// TwinCAT 3 PLC project KbRail
// ProgramVersion: 3.1.4022.7
// libraries:
//   Tc2_MC2, * (Beckhoff Automation GmbH)
//   Tc2_Standard, * (Beckhoff Automation GmbH)
//   Tc2_System, * (Beckhoff Automation GmbH)
//   Tc3_Module, * (Beckhoff Automation GmbH)
// project tree:
//   DUTs/ ST_AxisGroup.TcDUT
//   / PlcTask.TcTTO
//   POUs/ MAIN.TcPOU
// real-time tasks:
//   TASK PlcTask: cycle T#10ms, priority 20, ADS port 350
// motion (NC):
//   TASK NC-Task 1 SAF: cycle T#2ms, priority 4, ADS port 501
//   TASK NC-Task 1 SVB: cycle T#10ms, priority 8, ADS port 511
//   AXIS Axis 1 (id 1)
//     Dynamic: AccelerationMaximum=0.6, DecelerationMaximum=0.6, Acceleration=0.59988, Deceleration=0.59988, Jerk=1.19952, DelayTime=0.008
//     Velo: Maximum=0.1
//     OtherSettings: AllowMotionCmdToSlave=true
//     encoder EncType=29
//       EncPara: ScaleFactorNumerator=1e-06, MaxCount=#xffffffff, EvaluationDirection=2
//         SoftEndMinControl: Enable=true, Range=5
//         Inc: RefSoftSyncMask=#x0000ffff
//     drive DrvType=24
//       DrvPara: Inverse=true
//         Analog: VeloReferenz=0.4, ScaleFactorActTorque=0.1
//         TimeComp: TaskDelayCycles=1
//     controller CtrType=1
//       CtrPara: PriorControlFactor=1
//         PosDiffControl: Range=0.2
//         Observer: BandWidth=20
//   AXIS Axis 2 (id 2)
//     Dynamic: AccelerationMaximum=0.6, DecelerationMaximum=0.6, Acceleration=0.59988, Deceleration=0.59988, Jerk=1.19952, DelayTime=0.008
//     Velo: Maximum=0.1
//     OtherSettings: AllowMotionCmdToSlave=true
//     encoder EncType=29
//       EncPara: ScaleFactorNumerator=1e-06, MaxCount=#xffffffff
//         SoftEndMinControl: Enable=true, Range=5
//         Inc: RefSoftSyncMask=#x0000ffff
//     drive DrvType=24
//       DrvPara: Inverse=true
//         Analog: VeloReferenz=0.4, ScaleFactorActTorque=0.1
//         TimeComp: TaskDelayCycles=1
//     controller CtrType=1
//       CtrPara: PriorControlFactor=1
//         PosDiffControl: Range=0.2
//         Observer: BandWidth=20
//   AXIS Axis 3 (id 3)
//     General: UnitName=nm
//     Dynamic: AccelerationMaximum=0.6, DecelerationMaximum=0.6, Acceleration=0.59988, Deceleration=0.59988, Jerk=1.19952, DelayTime=0.008
//     Velo: Maximum=0.1
//     OtherSettings: AllowMotionCmdToSlave=true
//     encoder EncType=29
//       EncPara: ScaleFactorNumerator=1e-06, MaxCount=#xffffffff
//         SoftEndMinControl: Enable=true, Range=6.25
//         Inc: RefSoftSyncMask=#x0000ffff
//     drive DrvType=24
//       DrvPara: Inverse=true
//         Analog: VeloReferenz=0.4, ScaleFactorActTorque=0.1
//         TimeComp: TaskDelayCycles=1
//     controller CtrType=1
//       CtrPara: PriorControlFactor=1
//         PosDiffControl: Range=0.2
//         Observer: BandWidth=20
//   AXIS Axis 4 (id 4)
//     General: UnitName=nm
//     Dynamic: AccelerationMaximum=0.6, DecelerationMaximum=0.6, Acceleration=0.59988, Deceleration=0.59988, Jerk=1.19952, DelayTime=0.008
//     Velo: Maximum=1
//     OtherSettings: AllowMotionCmdToSlave=true
//     encoder EncType=29
//       EncPara: ScaleFactorNumerator=1e-06, MaxCount=#xffffffff
//         SoftEndMinControl: Enable=true, Range=5.5
//         Inc: RefSoftSyncMask=#x0000ffff
//     drive DrvType=24
//       DrvPara: Inverse=true
//         Analog: VeloReferenz=0.4, ScaleFactorActTorque=0.1
//         TimeComp: TaskDelayCycles=1
//     controller CtrType=1
//       CtrPara: PriorControlFactor=1
//         PosDiffControl: Range=0.2
//         Observer: BandWidth=20
// I/O:
//   DEVICE Device 1 (EtherCAT), AmsNetId 192.168.1.82.3.1
//     Term 12 (EK1100) [EK1100 EtherCAT Coupler (2A E-Bus)]
//       E1(EL7041) [EL7041 1Ch. Stepper motor output stage (50V, 5A)]
//       E2(EL5042) [EL5042 2Ch. BiSS-C Encoder]
//       E3(EL7041) [EL7041 1Ch. Stepper motor output stage (50V, 5A)]
//       E4(EL3202-0010)
//       E5(EL7041) [EL7041 1Ch. Stepper motor output stage (50V, 5A)]
//       E6(EL5042) [EL5042 2Ch. BiSS-C Encoder]
//       E7(EL7041) [EL7041 1Ch. Stepper motor output stage (50V, 5A)]
//       E8(EL3202-0010)
//       Term 23 (EL9011) [EL9011 End Terminal]
// variable links:
//   NC-Task 1 SAF/Axes/Axis 1 <-> Device 1 (EtherCAT)/Term 12 (EK1100)/E1(EL7041)
//     Drive/Inputs/In/nState1 @bit 3 <-> STM Status/Status/Error
//     Drive/Inputs/In/nState1 @bit 5 <-> STM Status/Status/Moving negative
//     Drive/Inputs/In/nState1 @bit 4 <-> STM Status/Status/Moving positive
//     Drive/Inputs/In/nState1 @bit 1 <-> STM Status/Status/Ready
//     Drive/Inputs/In/nState1 <-> STM Status/Status/Ready to enable
//     Drive/Inputs/In/nState1 @bit 6 <-> STM Status/Status/Torque reduced
//     Drive/Inputs/In/nState1 @bit 2 <-> STM Status/Status/Warning
//     Drive/Inputs/In/nState2 @bit 5 <-> STM Status/Status/Sync error
//     Drive/Inputs/In/nState2 @bit 7 <-> STM Status/Status/TxPDO Toggle
//     Drive/Inputs/In/nState4 @bit 1 <-> WcState/InputToggle
//     Drive/Inputs/In/nState4 <-> WcState/WcState
//     Drive/Outputs/Out/nCtrl1 <-> STM Control/Control/Enable
//     Drive/Outputs/Out/nCtrl1 @bit 2 <-> STM Control/Control/Reduce torque
//     Drive/Outputs/Out/nCtrl1 @bit 1 <-> STM Control/Control/Reset
//     Drive/Outputs/Out/nDataOut2[0] <-> STM Velocity/Velocity
//   NC-Task 1 SAF/Axes/Axis 1 <-> Device 1 (EtherCAT)/Term 12 (EK1100)/E2(EL5042)
//     Enc/Inputs/In/nComState @bit 1 <-> WcState/InputToggle
//     Enc/Inputs/In/nComState <-> WcState/WcState
//     Enc/Inputs/In/nDataIn1 <-> FB Inputs Channel 1/Position
//     Enc/Inputs/In/nState1 @bit 12 <-> FB Inputs Channel 1/Status/Diag
//     Enc/Inputs/In/nState1 @bit 1 <-> FB Inputs Channel 1/Status/Error
//     Enc/Inputs/In/nState1 @bit 14 <-> FB Inputs Channel 1/Status/Input cycle counter
//     Enc/Inputs/In/nState1 @bit 2 <-> FB Inputs Channel 1/Status/Ready
//     Enc/Inputs/In/nState1 @bit 13 <-> FB Inputs Channel 1/Status/TxPDO State
//     Enc/Inputs/In/nState1 <-> FB Inputs Channel 1/Status/Warning
//   NC-Task 1 SAF/Axes/Axis 2 <-> Device 1 (EtherCAT)/Term 12 (EK1100)/E2(EL5042)
//     Enc/Inputs/In/nComState @bit 1 <-> WcState/InputToggle
//     Enc/Inputs/In/nComState <-> WcState/WcState
//     Enc/Inputs/In/nDataIn1 <-> FB Inputs Channel 2/Position
//     Enc/Inputs/In/nState1 @bit 12 <-> FB Inputs Channel 2/Status/Diag
//     Enc/Inputs/In/nState1 @bit 1 <-> FB Inputs Channel 2/Status/Error
//     Enc/Inputs/In/nState1 @bit 14 <-> FB Inputs Channel 2/Status/Input cycle counter
//     Enc/Inputs/In/nState1 @bit 2 <-> FB Inputs Channel 2/Status/Ready
//     Enc/Inputs/In/nState1 @bit 13 <-> FB Inputs Channel 2/Status/TxPDO State
//     Enc/Inputs/In/nState1 <-> FB Inputs Channel 2/Status/Warning
//   NC-Task 1 SAF/Axes/Axis 2 <-> Device 1 (EtherCAT)/Term 12 (EK1100)/E3(EL7041)
//     Drive/Inputs/In/nState1 @bit 3 <-> STM Status/Status/Error
//     Drive/Inputs/In/nState1 @bit 5 <-> STM Status/Status/Moving negative
//     Drive/Inputs/In/nState1 @bit 4 <-> STM Status/Status/Moving positive
//     Drive/Inputs/In/nState1 @bit 1 <-> STM Status/Status/Ready
//     Drive/Inputs/In/nState1 <-> STM Status/Status/Ready to enable
//     Drive/Inputs/In/nState1 @bit 6 <-> STM Status/Status/Torque reduced
//     Drive/Inputs/In/nState1 @bit 2 <-> STM Status/Status/Warning
//     Drive/Inputs/In/nState2 @bit 5 <-> STM Status/Status/Sync error
//     Drive/Inputs/In/nState2 @bit 7 <-> STM Status/Status/TxPDO Toggle
//     Drive/Inputs/In/nState4 @bit 1 <-> WcState/InputToggle
//     Drive/Inputs/In/nState4 <-> WcState/WcState
//     Drive/Outputs/Out/nCtrl1 <-> STM Control/Control/Enable
//     Drive/Outputs/Out/nCtrl1 @bit 2 <-> STM Control/Control/Reduce torque
//     Drive/Outputs/Out/nCtrl1 @bit 1 <-> STM Control/Control/Reset
//     Drive/Outputs/Out/nDataOut2[0] <-> STM Velocity/Velocity
//   NC-Task 1 SAF/Axes/Axis 3 <-> Device 1 (EtherCAT)/Term 12 (EK1100)/E5(EL7041)
//     Drive/Inputs/In/nState1 @bit 3 <-> STM Status/Status/Error
//     Drive/Inputs/In/nState1 @bit 5 <-> STM Status/Status/Moving negative
//     Drive/Inputs/In/nState1 @bit 4 <-> STM Status/Status/Moving positive
//     Drive/Inputs/In/nState1 @bit 1 <-> STM Status/Status/Ready
//     Drive/Inputs/In/nState1 <-> STM Status/Status/Ready to enable
//     Drive/Inputs/In/nState1 @bit 6 <-> STM Status/Status/Torque reduced
//     Drive/Inputs/In/nState1 @bit 2 <-> STM Status/Status/Warning
//     Drive/Inputs/In/nState2 @bit 5 <-> STM Status/Status/Sync error
//     Drive/Inputs/In/nState2 @bit 7 <-> STM Status/Status/TxPDO Toggle
//     Drive/Inputs/In/nState4 @bit 1 <-> WcState/InputToggle
//     Drive/Inputs/In/nState4 <-> WcState/WcState
//     Drive/Outputs/Out/nCtrl1 <-> STM Control/Control/Enable
//     Drive/Outputs/Out/nCtrl1 @bit 2 <-> STM Control/Control/Reduce torque
//     Drive/Outputs/Out/nCtrl1 @bit 1 <-> STM Control/Control/Reset
//     Drive/Outputs/Out/nDataOut2[0] <-> STM Velocity/Velocity
//   NC-Task 1 SAF/Axes/Axis 3 <-> Device 1 (EtherCAT)/Term 12 (EK1100)/E6(EL5042)
//     Enc/Inputs/In/nComState @bit 1 <-> WcState/InputToggle
//     Enc/Inputs/In/nComState <-> WcState/WcState
//     Enc/Inputs/In/nDataIn1 <-> FB Inputs Channel 1/Position
//     Enc/Inputs/In/nState1 @bit 12 <-> FB Inputs Channel 1/Status/Diag
//     Enc/Inputs/In/nState1 @bit 1 <-> FB Inputs Channel 1/Status/Error
//     Enc/Inputs/In/nState1 @bit 14 <-> FB Inputs Channel 1/Status/Input cycle counter
//     Enc/Inputs/In/nState1 @bit 2 <-> FB Inputs Channel 1/Status/Ready
//     Enc/Inputs/In/nState1 @bit 13 <-> FB Inputs Channel 1/Status/TxPDO State
//     Enc/Inputs/In/nState1 <-> FB Inputs Channel 1/Status/Warning
//   NC-Task 1 SAF/Axes/Axis 4 <-> Device 1 (EtherCAT)/Term 12 (EK1100)/E6(EL5042)
//     Enc/Inputs/In/nComState @bit 1 <-> WcState/InputToggle
//     Enc/Inputs/In/nComState <-> WcState/WcState
//     Enc/Inputs/In/nDataIn1 <-> FB Inputs Channel 2/Position
//     Enc/Inputs/In/nState1 @bit 12 <-> FB Inputs Channel 2/Status/Diag
//     Enc/Inputs/In/nState1 @bit 1 <-> FB Inputs Channel 2/Status/Error
//     Enc/Inputs/In/nState1 @bit 14 <-> FB Inputs Channel 2/Status/Input cycle counter
//     Enc/Inputs/In/nState1 @bit 2 <-> FB Inputs Channel 2/Status/Ready
//     Enc/Inputs/In/nState1 @bit 13 <-> FB Inputs Channel 2/Status/TxPDO State
//     Enc/Inputs/In/nState1 <-> FB Inputs Channel 2/Status/Warning
//   NC-Task 1 SAF/Axes/Axis 4 <-> Device 1 (EtherCAT)/Term 12 (EK1100)/E7(EL7041)
//     Drive/Inputs/In/nState1 @bit 3 <-> STM Status/Status/Error
//     Drive/Inputs/In/nState1 @bit 5 <-> STM Status/Status/Moving negative
//     Drive/Inputs/In/nState1 @bit 4 <-> STM Status/Status/Moving positive
//     Drive/Inputs/In/nState1 @bit 1 <-> STM Status/Status/Ready
//     Drive/Inputs/In/nState1 <-> STM Status/Status/Ready to enable
//     Drive/Inputs/In/nState1 @bit 6 <-> STM Status/Status/Torque reduced
//     Drive/Inputs/In/nState1 @bit 2 <-> STM Status/Status/Warning
//     Drive/Inputs/In/nState2 @bit 5 <-> STM Status/Status/Sync error
//     Drive/Inputs/In/nState2 @bit 7 <-> STM Status/Status/TxPDO Toggle
//     Drive/Inputs/In/nState4 @bit 1 <-> WcState/InputToggle
//     Drive/Inputs/In/nState4 <-> WcState/WcState
//     Drive/Outputs/Out/nCtrl1 <-> STM Control/Control/Enable
//     Drive/Outputs/Out/nCtrl1 @bit 2 <-> STM Control/Control/Reduce torque
//     Drive/Outputs/Out/nCtrl1 @bit 1 <-> STM Control/Control/Reset
//     Drive/Outputs/Out/nDataOut2[0] <-> STM Velocity/Velocity
//   KbRail/KbRail Instance <-> Device 1 (EtherCAT)/Term 12 (EK1100)/E1(EL7041)
//     PlcTask Inputs/MAIN.M[1].bLimHigh <-> STM Status/Status/Digital input 1
//     PlcTask Inputs/MAIN.M[1].bLimLow <-> STM Status/Status/Digital input 2
//   KbRail/KbRail Instance <-> Device 1 (EtherCAT)/Term 12 (EK1100)/E3(EL7041)
//     PlcTask Inputs/MAIN.M[2].bLimHigh <-> STM Status/Status/Digital input 1
//     PlcTask Inputs/MAIN.M[2].bLimLow <-> STM Status/Status/Digital input 2
//   KbRail/KbRail Instance <-> Device 1 (EtherCAT)/Term 12 (EK1100)/E4(EL3202-0010)
//     PlcTask Inputs/MAIN.RTD[1] <-> RTD Inputs Channel 1/Value
//     PlcTask Inputs/MAIN.RTD[2] <-> RTD Inputs Channel 2/Value
//   KbRail/KbRail Instance <-> Device 1 (EtherCAT)/Term 12 (EK1100)/E5(EL7041)
//     PlcTask Inputs/MAIN.M[3].bLimHigh <-> STM Status/Status/Digital input 1
//     PlcTask Inputs/MAIN.M[3].bLimLow <-> STM Status/Status/Digital input 2
//   KbRail/KbRail Instance <-> Device 1 (EtherCAT)/Term 12 (EK1100)/E7(EL7041)
//     PlcTask Inputs/MAIN.M[4].bLimHigh <-> STM Status/Status/Digital input 1
//     PlcTask Inputs/MAIN.M[4].bLimLow <-> STM Status/Status/Digital input 2
//   KbRail/KbRail Instance <-> Device 1 (EtherCAT)/Term 12 (EK1100)/E8(EL3202-0010)
//     PlcTask Inputs/MAIN.RTD[3] <-> RTD Inputs Channel 1/Value
//     PlcTask Inputs/MAIN.RTD[4] <-> RTD Inputs Channel 2/Value
//   KbRail/KbRail Instance <-> NC-Task 1 SAF/Axes/Axis 1
//     PlcTask Inputs/MAIN.M[1].axisRef.NcToPlc <-> Outputs/ToPlc
//     PlcTask Outputs/MAIN.M[1].axisRef.PlcToNc <-> Inputs/FromPlc
//   KbRail/KbRail Instance <-> NC-Task 1 SAF/Axes/Axis 2
//     PlcTask Inputs/MAIN.M[2].axisRef.NcToPlc <-> Outputs/ToPlc
//     PlcTask Outputs/MAIN.M[2].axisRef.PlcToNc <-> Inputs/FromPlc
//   KbRail/KbRail Instance <-> NC-Task 1 SAF/Axes/Axis 3
//     PlcTask Inputs/MAIN.M[3].axisRef.NcToPlc <-> Outputs/ToPlc
//     PlcTask Outputs/MAIN.M[3].axisRef.PlcToNc <-> Inputs/FromPlc
//   KbRail/KbRail Instance <-> NC-Task 1 SAF/Axes/Axis 4
//     PlcTask Inputs/MAIN.M[4].axisRef.NcToPlc <-> Outputs/ToPlc
//     PlcTask Outputs/MAIN.M[4].axisRef.PlcToNc <-> Inputs/FromPlc

CONFIGURATION KbRail
    RESOURCE PLC ON TwinCAT3
        TASK PlcTask(INTERVAL := T#10ms, PRIORITY := 20);
        PROGRAM MAIN WITH PlcTask : MAIN;
    END_RESOURCE
END_CONFIGURATION

// ---- DUTs/ST_AxisGroup.TcDUT
TYPE ST_AxisGroup :
STRUCT
	//basic built in functions
	mcPower		: MC_Power;
	mcReset		: MC_Reset;
	mcMoveAbs	: MC_MoveAbsolute;
	mcMoveRel	: MC_MoveRelative;
	mcHome		: MC_Home;
	mcStop		: MC_Stop;
	mcJog		: MC_Jog;
	
	//linkable variables
	axisRef				: AXIS_REF;;
	bLimHigh 	AT %I*	: BOOL;
	bLimLow 	AT %I*	: BOOL;

END_STRUCT
END_TYPE

// ---- POUs/MAIN.TcPOU
PROGRAM MAIN
VAR
	{attribute 'TcLinkTo' := '	[1].bLimHigh	:=	TIID^Device 1 (EtherCAT)^Term 12 (EK1100)^E1(EL7041)^STM Status^Status^Digital input 1;
								[1].bLimLow		:=	TIID^Device 1 (EtherCAT)^Term 12 (EK1100)^E1(EL7041)^STM Status^Status^Digital input 2;
								[2].bLimHigh	:=	TIID^Device 1 (EtherCAT)^Term 12 (EK1100)^E3(EL7041)^STM Status^Status^Digital input 1;
								[2].bLimLow		:=	TIID^Device 1 (EtherCAT)^Term 12 (EK1100)^E3(EL7041)^STM Status^Status^Digital input 2;
								[3].bLimHigh	:=	TIID^Device 1 (EtherCAT)^Term 12 (EK1100)^E5(EL7041)^STM Status^Status^Digital input 1;
								[3].bLimLow		:=	TIID^Device 1 (EtherCAT)^Term 12 (EK1100)^E5(EL7041)^STM Status^Status^Digital input 2;
								[4].bLimHigh	:=	TIID^Device 1 (EtherCAT)^Term 12 (EK1100)^E7(EL7041)^STM Status^Status^Digital input 1;
								[4].bLimLow		:=	TIID^Device 1 (EtherCAT)^Term 12 (EK1100)^E7(EL7041)^STM Status^Status^Digital input 2'}
	M			: ARRAY [1 .. 4] OF ST_AxisGroup;
	
	{attribute 'TcLinkTo' := '	[1]	:=	TIID^Device 1 (EtherCAT)^Term 12 (EK1100)^E4(EL3202-0010)^RTD Inputs Channel 1^Value;
								[2]	:=	TIID^Device 1 (EtherCAT)^Term 12 (EK1100)^E4(EL3202-0010)^RTD Inputs Channel 2^Value;
								[3]	:=	TIID^Device 1 (EtherCAT)^Term 12 (EK1100)^E8(EL3202-0010)^RTD Inputs Channel 1^Value;
								[4]	:=	TIID^Device 1 (EtherCAT)^Term 12 (EK1100)^E8(EL3202-0010)^RTD Inputs Channel 2^Value'}
	RTD AT %I*	: ARRAY [1 .. 4] OF INT;
	
	
END_VAR

(*update Axis_Ref status*)
M[1].axisRef.ReadStatus();
M[2].axisRef.ReadStatus();
M[3].axisRef.ReadStatus();
M[4].axisRef.ReadStatus();

(*Enable motors*)
M[1].mcPower(Axis:=M[1].axisRef, Enable:=TRUE, Enable_Positive:=M[1].bLimHigh, Enable_Negative:=M[1].bLimLow);
M[2].mcPower(Axis:=M[2].axisRef, Enable:=TRUE, Enable_Positive:=M[2].bLimHigh, Enable_Negative:=M[2].bLimLow);
M[3].mcPower(Axis:=M[3].axisRef, Enable:=TRUE, Enable_Positive:=M[3].bLimHigh, Enable_Negative:=M[3].bLimLow);
M[4].mcPower(Axis:=M[4].axisRef, Enable:=TRUE, Enable_Positive:=M[4].bLimHigh, Enable_Negative:=M[4].bLimLow);

END_PROGRAM
